{attribute 'GeneratedUsingTerminal: IODEVICETYPE_ETHERCATPROT'}
{attribute addProperty BoxType "IODEVICETYPE_ETHERCATPROT"}
{attribute addProperty Id "Beckhoff_EQ1xxxBeckhoff_EQ1xxx_F67C323D78Beckhoff_EQ2xxxBeckhoff_EQ2xxx_A19B669C247Beckhoff_EQ3xxxBeckhoff_EQ3xxx_0F87BCE2718SyncUnitsSyncUnits_99E584AF18InputsInputs_25A0042B160OutputsOutputs_2397A10E106InfoDataInfoData_E68C61CD28"}
{attribute addProperty CRC "2798911577"}
{attribute addProperty Size "1355"}
TYPE EtherCAT_Master_EQxxxx_A6D40059 :
STRUCT
	{attribute addProperty Name "Beckhoff_EQ1xxx"}
	{attribute addProperty PreviousPort "EtherCAT_Master_EQxxxx : Master"}
	Beckhoff_EQ1xxx : Beckhoff_EQ1xxx_F67C323D;
	{attribute addProperty Name "Beckhoff_EQ2xxx"}
	{attribute addProperty PreviousPort "Beckhoff EQ1xxx : C"}
	Beckhoff_EQ2xxx : Beckhoff_EQ2xxx_A19B669C;
	{attribute addProperty Name "Beckhoff_EQ3xxx"}
	{attribute addProperty PreviousPort "Beckhoff EQ2xxx : C"}
	Beckhoff_EQ3xxx : Beckhoff_EQ3xxx_0F87BCE2;
	{attribute addProperty Name "SyncUnits"}
	SyncUnits : SyncUnits_99E584AF;
	{attribute addProperty Name "Inputs"}
	Inputs : Inputs_25A0042B;
	{attribute addProperty Name "Outputs"}
	Outputs : Outputs_2397A10E;
	{attribute addProperty Name "InfoData"}
	InfoData : InfoData_E68C61CD;
END_STRUCT
END_TYPE

(* stored: Version 1.2.0.0, ProductVersion 3.1.4024.9
   DUT EtherCAT_Master_EQxxxx_A6D40059: Id {44110839-7bb8-44e2-b4e6-e933b857cf04} *)
